FUNCTION_BLOCK DiagServer0 (* Sends sensor data and diagnostic data over a network. Wrapper for a SERVER function block. *)
  (* Standard: 61499-2; Description: A client can request diagnostic data from this function block. *)
  (* Version 1.0, 2017-08-27, Marc Jakobi, HTW Berlin *)
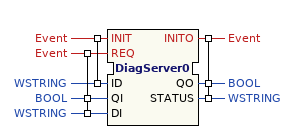
  EVENT_INPUT
    INIT WITH ID; (* Initialization Request *)
    REQ WITH DI, QI; (* Normal Execution Request *)
  END_EVENT
  EVENT_OUTPUT
    INITO WITH QO, STATUS; (* Initialization Confirm *)
  END_EVENT
  VAR_INPUT
    ID : WSTRING; (* Connection identifier *)
    QI : BOOL; (* Diagnostic qualifier *)
    DI : WSTRING; (* Diagnostic info *)
  END_VAR
  VAR_OUTPUT
    QO : BOOL; (* Output event qualifier *)
    STATUS : WSTRING; (* Service status *)
  END_VAR
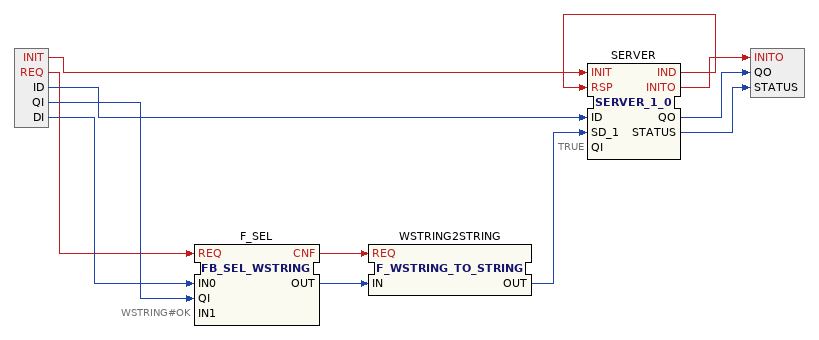
  FBS
    WSTRING2STRING : F_WSTRING_TO_STRING;
    SERVER : SERVER_1_0(QI := TRUE);
    F_SEL : FB_SEL_WSTRING(IN1 := WSTRING#OK);
  END_FBS
  EVENT_CONNECTIONS
    INIT TO SERVER.INIT;
    SERVER.IND TO SERVER.RSP;
    SERVER.INITO TO INITO;
    REQ TO F_SEL.REQ;
    F_SEL.CNF TO WSTRING2STRING.REQ;
  END_CONNECTIONS
  DATA_CONNECTIONS
    ID TO SERVER.ID;
    WSTRING2STRING.OUT TO SERVER.SD_1;
    SERVER.QO TO QO;
    SERVER.STATUS TO STATUS;
    DI TO F_SEL.IN0;
    F_SEL.OUT TO WSTRING2STRING.IN;
    QI TO F_SEL.QI;
  END_CONNECTIONS
END_FUNCTION_BLOCK
